Fanuc KAREL source: kf00100.KL

-- PROVISIONAL review KL for V940-1; original PC SHA256 d4992831918aef230a8aea4e0757574bc75ef93169d523a8747936748dd8e3f1
-- Incomplete behavior may be omitted. Consult companion uncertainty JSON. Do not deploy.
PROGRAM KF00100
%NOLOCKGROUP
BEGIN
  -- V9_ZERO_TABLE_METADATA_HINT layout=0002_ascii; no indexed target words; source/name/runtime held
  -- UNRESOLVED_PC offsets 5-16; opcodes 2E,23
  -- UNRESOLVED_PC offsets 21-32; opcodes 2E,23
  -- UNRESOLVED_PC offsets 37-63; opcodes 27,27,9D,22,1C,22,27,9D,31
  -- UNRESOLVED_PC offsets 68-72; opcodes 7F
END KF00100
